(* LS Electric XG5000 project: AC1duobleanaloge *)
(* PLC NewPLC *)
(* module base 0 slot 0: Input/Output Module:XEC-DR60S (DC 24V INPUT 36points/RELAY OUTPUT 24points) *)
(* module base 0 slot 1: Input/Output Module:XBE-DR16A (DC 24V INPUT/RELAY OUTPUT, 16points) *)
(* module base 0 slot 2: Analog IO Module:XBF-AH04A (I/O, 2/2 CH) *)
(* module base 0 slot 9: Analog Output Module:XBO-DA02A (Volt/Current, 2-CH) *)
(* module base 0 slot 10: Analog Output Module:XBO-DA02A (Volt/Current, 2-CH) *)
VAR_GLOBAL
    _02_DA0_ACT AT %UX0.2.18 : BOOL; (* Analog IO Module: Output CH0 Active *)
    _02_DA0_DATA AT %UW0.2.7 : WORD; (* Analog IO Module: Output CH0 DATA *)
    _02_DA0_OUTEN AT %UX0.2.96 : BOOL; (* Analog IO Module: Output CH0 Status Setting *)
    _02_DA1_ACT AT %UX0.2.19 : BOOL; (* Analog IO Module: Output CH1 Active *)
    _02_DA1_DATA AT %UW0.2.8 : WORD; (* Analog IO Module: Output CH1 DATA *)
    _02_DA1_OUTEN AT %UX0.2.97 : BOOL; (* Analog IO Module: Output CH1 Status Setting *)
    _09_DA0_ACT AT %UX0.9.18 : BOOL; (* Analog Output Option Board: Output CH0 Active *)
    _09_DA0_OUTEN AT %UX0.9.96 : BOOL; (* Analog Output Option Board: Output CH0 Status Setting *)
    _09_DA1_ACT AT %UX0.9.19 : BOOL; (* Analog Output Option Board: Output CH1 Active *)
    _09_DA1_OUTEN AT %UX0.9.97 : BOOL; (* Analog Output Option Board: Output CH1 Status Setting *)
    _0A_DA0_ACT AT %UX0.10.18 : BOOL; (* Analog Output Option Board: Output CH0 Active *)
    _0A_DA0_OUTEN AT %UX0.10.96 : BOOL; (* Analog Output Option Board: Output CH0 Status Setting *)
    _0A_DA1_ACT AT %UX0.10.19 : BOOL; (* Analog Output Option Board: Output CH1 Active *)
    _0A_DA1_OUTEN AT %UX0.10.97 : BOOL; (* Analog Output Option Board: Output CH1 Status Setting *)
END_VAR

PROGRAM NewProgram_Copy (* task: Scan Program *)
VAR
    AAAA : WORD;
    aaaaaaaaaaaaaaa : REAL;
    acCONTROL AT %IX0.0.0 : BOOL;
    ACTRANS : BOOL;
    ADD1 : WORD;
    ADD2 : WORD;
    ANDOUT1 : WORD;
    AUTO AT %MX1 : BOOL;
    autoinhibit AT %MX222 : BOOL;
    BLOCK : UINT;
    chillerready : BOOL;
    COMPRESSOR : BOOL;
    CONTACTOR1 AT %QX0.0.0 : BOOL;
    CONTACTOR10 AT %QX0.0.9 : BOOL;
    CONTACTOR11 AT %QX0.0.20 : BOOL;
    CONTACTOR110 AT %IX0.0.29 : BOOL;
    CONTACTOR12 AT %QX0.0.21 : BOOL;
    CONTACTOR120 AT %IX0.0.30 : BOOL;
    CONTACTOR13 AT %QX0.0.22 : BOOL;
    CONTACTOR130 AT %IX0.0.31 : BOOL;
    CONTACTOR14 AT %QX0.0.23 : BOOL;
    CONTACTOR140 AT %IX0.0.32 : BOOL;
    CONTACTOR15 AT %QX0.1.0 : BOOL;
    CONTACTOR150 AT %IX0.0.33 : BOOL;
    CONTACTOR16 AT %QX0.1.1 : BOOL;
    CONTACTOR160 AT %IX0.0.34 : BOOL;
    CONTACTOR17 AT %QX0.1.2 : BOOL;
    CONTACTOR170 AT %IX0.1.1 : BOOL;
    CONTACTOR18 AT %QX0.1.3 : BOOL;
    CONTACTOR180 AT %IX0.1.0 : BOOL;
    CONTACTOR2 AT %QX0.0.1 : BOOL;
    CONTACTOR3 AT %QX0.0.2 : BOOL;
    CONTACTOR4 AT %QX0.0.3 : BOOL;
    CONTACTOR5 AT %QX0.0.4 : BOOL;
    CONTACTOR6 AT %QX0.0.5 : BOOL;
    CONTACTOR7 AT %QX0.0.6 : BOOL;
    CONTACTOR8 AT %QX0.0.7 : BOOL;
    CONTACTOR9 AT %QX0.0.8 : BOOL;
    CV : INT;
    damperon : BOOL;
    dcpower AT %IX0.0.1 : BOOL;
    DCPOWERK AT %QX0.1.4 : BOOL;
    dcpowerman AT %MX18 : BOOL;
    ddddddd : BOOL;
    DIV11 : WORD;
    DIV12 : INT;
    DIV124 : INT;
    DIV2 : WORD;
    DIV21 : WORD;
    DIV22 : WORD;
    DIV23 : WORD;
    DIV32 : INT;
    DIV33 : INT;
    DOOR1 AT %IX0.1.6 : BOOL;
    DOOR2 AT %IX0.1.7 : BOOL;
    DRIVE1ALARM AT %MX420 : BOOL;
    DRIVE2ALARM AT %MX421 : BOOL;
    DRIVEK1 AT %MX90 : BOOL;
    DRIVEK2 AT %MX91 : BOOL;
    DRIVEK3 : BOOL;
    DRIVEK4 : BOOL;
    DRIVEK5 : BOOL;
    DRIVEK6 : BOOL;
    DRIVEPUMP AT %MX92 : BOOL;
    dvi2 : DWORD;
    E11 : WORD;
    E2 : WORD;
    EE : WORD;
    EE1 : WORD;
    EE2 : WORD;
    ERR : BOOL;
    ET : TIME;
    FANREFSCALE : WORD;
    FANRUN : BOOL;
    FILTERRUN AT %MX50 : BOOL;
    FR10 AT %IX0.0.23 : BOOL;
    FR11 AT %IX0.0.24 : BOOL;
    FR12 AT %IX0.0.25 : BOOL;
    FR13 AT %IX0.0.26 : BOOL;
    FR14 AT %IX0.0.27 : BOOL;
    FR15 AT %IX0.0.28 : BOOL;
    FR8 AT %IX0.0.21 : BOOL;
    FR9 AT %IX0.0.22 : BOOL;
    HIMIDITYSCAL2 : WORD;
    HUMID2 : WORD;
    HUMID3 : WORD;
    HUMID4 : BOOL;
    HUMID5 : BOOL;
    HUMIDHIVALUE1 : WORD;
    HUMIDITIERR1 : WORD;
    HUMIDITYOUTSCAL : WORD;
    HUMIDLOWLIM1 : WORD;
    HUMIDNO1 : BOOL;
    HUMIDON : BOOL;
    hummidd : WORD;
    IN1 : SINT;
    IN10 : WORD;
    incin : WORD;
    inhumreal : REAL;
    inhumreal1 : REAL;
    inrealhuscale : REAL;
    inrealhuscale1 : REAL;
    INST : TON;
    INST1 : TON;
    INST10 : PIDRUN;
    INST11 : PIDRUN;
    INST12 : TON_UINT;
    INST13 : TON_UINT;
    INST14 : TON;
    INST15 : TON;
    INST16 : TON;
    INST17 : TON;
    INST18 : TON;
    INST19 : TON;
    INST2 : TON;
    INST20 : TON;
    INST21 : TON;
    INST22 : TON;
    INST23 : TON;
    INST24 : TON;
    INST25 : TON;
    INST26 : CTU_INT;
    INST27 : TON;
    INST28 : TON;
    INST29 : CTU_INT;
    INST3 : TON;
    INST30 : TON;
    INST31 : TON;
    INST32 : TON;
    INST33 : TON;
    INST34 : TON;
    INST35 : TON;
    INST36 : TON;
    INST37 : CTU_INT;
    INST38 : CTU_INT;
    INST39 : TON;
    INST4 : TON;
    INST40 : TON_UINT;
    INST41 : TON_UINT;
    INST42 : TON_UINT;
    INST43 : TON_UINT;
    INST44 : TON_UINT;
    INST45 : TON_UINT;
    INST46 : TON_UINT;
    INST47 : TMR;
    INST48 : TON_UINT;
    INST49 : TON_UINT;
    INST5 : TON;
    INST50 : TON_UINT;
    INST51 : TON_UINT;
    INST52 : TON_UINT;
    INST53 : TON;
    INST54 : TON;
    INST55 : TON;
    INST56 : TON;
    INST57 : TON;
    INST58 : TON;
    INST59 : TON;
    INST6 : TON;
    INST60 : TON;
    INST61 : TON;
    INST62 : CTU_INT;
    INST63 : CTR;
    INST64 : TON;
    INST65 : TON;
    INST66 : TON;
    INST67 : TON;
    INST68 : TON;
    INST69 : TON;
    INST7 : TON;
    INST70 : TON;
    INST71 : TON;
    INST72 : TON;
    INST73 : TON;
    INST74 : TON;
    INST75 : TON;
    INST76 : TON;
    INST77 : TON;
    INST8 : TON;
    INST9 : TON;
    K10ENDIS AT %MX129 : BOOL;
    K1B AT %MX95 : BOOL;
    k1endis AT %MX120 : BOOL;
    K2B AT %MX97 : BOOL;
    k2ENDIS AT %MX121 : BOOL;
    K3B : BOOL;
    K3ENDIS AT %MX122 : BOOL;
    K4B : BOOL;
    K4ENDIS AT %MX123 : BOOL;
    K5B : BOOL;
    K5ENDIS AT %MX124 : BOOL;
    K6B : BOOL;
    K6ENDIS AT %MX125 : BOOL;
    K7ENDIS AT %MX126 : BOOL;
    K8ENDIS AT %MX127 : BOOL;
    K9ENDIS AT %MX128 : BOOL;
    KDISCH1 AT %MX96 : BOOL;
    KDISCH2 : BOOL;
    KDISCH3 : BOOL;
    KSUC AT %MX94 : BOOL;
    KSUC2 : BOOL;
    KSUC3 : BOOL;
    LOOP : UINT;
    man1 : BOOL;
    man10 : BOOL;
    man2 : BOOL;
    man3 : BOOL;
    man4 : BOOL;
    man5 : BOOL;
    man6 : BOOL;
    man7 : BOOL;
    man8 : BOOL;
    man9 : BOOL;
    mot1 : BOOL;
    mot10 : BOOL;
    mot11 : BOOL;
    mot12 : BOOL;
    mot2 : BOOL;
    mot3 : BOOL;
    mot4 : BOOL;
    mot5 : BOOL;
    mot6 : BOOL;
    mot7 : BOOL;
    mot8 : BOOL;
    mot9 : BOOL;
    motor10 : BOOL;
    motor11 : BOOL;
    motor12 : BOOL;
    motor13 : BOOL;
    motor9 : BOOL;
    ooot : INT;
    OUT : SINT;
    OUT10 : INT;
    OUT100 : INT;
    OUT101 : REAL;
    OUT102 : REAL;
    OUT103 : INT;
    OUT104 : WORD;
    OUT20 : INT;
    OUT200 : WORD;
    out201 : INT;
    OUT202 : WORD;
    OUT203 : INT;
    OUT21 : INT;
    OUT300 : REAL;
    OUT301 : REAL;
    out310 : REAL;
    OUT351 : REAL;
    OUT352 : REAL;
    OUT50 : WORD;
    OUT6 : WORD;
    OUT6bit : BOOL;
    outhumreal : REAL;
    OUTrealhuscale : REAL;
    OUTTMP : WORD;
    OUTTMPLOWLIM : WORD;
    ouuu : INT;
    ouuuuuuut : DWORD;
    PID_STAT : WORD;
    PUMPON : BOOL;
    Q : BOOL;
    rstauto AT %MX2 : BOOL;
    RUNOK AT %MX98 : BOOL;
    scal11 : REAL;
    scale22 : REAL;
    scale23 : REAL;
    setauto AT %MX0 : BOOL;
    STATE1 : BOOL;
    STATE2 : BOOL;
    STATE3 : BOOL;
    STATE4 : BOOL;
    STATE5 : BOOL;
    STATE6 : BOOL;
    STATE7 : BOOL;
    step1 : BOOL;
    step10 : BOOL;
    step2 : BOOL;
    step3 : BOOL;
    step4 : BOOL;
    step5 : BOOL;
    step6 : BOOL;
    step7 : BOOL;
    step8 : BOOL;
    step9 : BOOL;
    SUCTION1RUN : BOOL;
    SUMMER : BOOL;
    teee : INT;
    TEMPE11 : WORD;
    TEMPLOWLIM1 : WORD;
    TEMPLOWLIM2 : INT;
    TEMPMAX1 : WORD;
    TEMPMAX2 : INT;
    VALVEACPOWER AT %QX0.1.7 : BOOL;
    VFD1 AT %QX0.0.10 : BOOL;
    VFD10 AT %QX0.0.19 : BOOL;
    VFD2 AT %QX0.0.11 : BOOL;
    VFD3 AT %QX0.0.12 : BOOL;
    VFD4 AT %QX0.0.13 : BOOL;
    VFD5 AT %QX0.0.14 : BOOL;
    VFD6 AT %QX0.0.15 : BOOL;
    VFD7 AT %QX0.0.16 : BOOL;
    VFD8 AT %QX0.0.17 : BOOL;
    VFD9 AT %QX0.0.18 : BOOL;
    WINTER : BOOL;
END_VAR
VAR RETAIN
    coldtemp AT %WW400 : INT;
    COLDTMP AT %WW240 : WORD;
    DIFFMAX AT %WW144 : WORD;
    DIFFMIN AT %WW142 : WORD;
    DIV1 : WORD;
    E1 AT %WW2004 : WORD;
    fanspeedhilim AT %WW156 : WORD;
    fanspeedlowlim AT %WW158 : WORD;
    FRESHDAMPER AT %WW310 : WORD;
    HIMIDITYSCALOUT AT %WW2016 : WORD;
    HOTTEMP AT %WW402 : INT;
    HOTTMP AT %WW230 : WORD;
    HUMIDHIVALUE AT %WW2012 : WORD;
    HUMIDINLEFTSENSOR AT %WW190 : WORD;
    HUMIDINRIGHTSENSOR AT %WW186 : WORD;
    HUMIDITIERR AT %WW2010 : WORD;
    HUMIDLOWLIM AT %WW2014 : WORD;
    HUMOUTSENSOR AT %WW184 : WORD;
    HUMSUM AT %WW178 : WORD;
    INHUMIDOFSET AT %WW177 : WORD;
    INHUMIDYSCALE AT %WW200 : WORD;
    INHUMIDYSCALE1 AT %WW204 : WORD;
    LEFTHUMIDSV AT %WW302 : WORD;
    MEANTEMP AT %WW520 : WORD;
    money AT %WW2800 : WORD;
    OUT5 AT %WW2008 : WORD;
    OUTHUMIDOFSET AT %WW179 : WORD;
    OUTHUMIDYSCALE AT %WW202 : WORD;
    OUTTEMP AT %WW210 : INT;
    pump1refrence AT %WW50 : WORD;
    pump2refrence AT %WW51 : WORD;
    rightHUMIDSV AT %WW300 : WORD;
    RIGHTZONFANREF AT %WW250 : WORD;
    scale1 AT %WD379 : REAL;
    scale2 AT %WD377 : REAL;
    SCALE21 AT %WD387 : REAL;
    temmmp AT %WW444 : WORD;
    TEMPE1 AT %WW2006 : WORD;
    TEMPINLEFTSENSOR AT %WW188 : WORD;
    TEMPINRIGHTSENSOR AT %WW185 : WORD;
    TEMPLOWLIM AT %WW2002 : INT;
    TEMPMAX AT %WW2000 : INT;
    TEMPOUTSESOR AT %WW183 : WORD;
    TEMPPV AT %WW220 : INT;
    TEMPPV1 AT %WW224 : INT;
    TEMPSV AT %WW10 : WORD;
    TEMPSV1 AT %WW12 : WORD;
    time1 AT %WW880 : WORD;
    timeout AT %WW890 : WORD;
END_VAR
VAR_EXTERNAL
    _02_DA0_ACT : BOOL; (* AT %UX0.2.18 *) (* Analog IO Module: Output CH0 Active *)
    _02_DA0_DATA : WORD; (* AT %UW0.2.7 *) (* Analog IO Module: Output CH0 DATA *)
    _02_DA0_OUTEN : BOOL; (* AT %UX0.2.96 *) (* Analog IO Module: Output CH0 Status Setting *)
    _02_DA1_ACT : BOOL; (* AT %UX0.2.19 *) (* Analog IO Module: Output CH1 Active *)
    _02_DA1_DATA : WORD; (* AT %UW0.2.8 *) (* Analog IO Module: Output CH1 DATA *)
    _02_DA1_OUTEN : BOOL; (* AT %UX0.2.97 *) (* Analog IO Module: Output CH1 Status Setting *)
    _09_DA0_ACT : BOOL; (* AT %UX0.9.18 *) (* Analog Output Option Board: Output CH0 Active *)
    _09_DA0_OUTEN : BOOL; (* AT %UX0.9.96 *) (* Analog Output Option Board: Output CH0 Status Setting *)
    _09_DA1_ACT : BOOL; (* AT %UX0.9.19 *) (* Analog Output Option Board: Output CH1 Active *)
    _09_DA1_OUTEN : BOOL; (* AT %UX0.9.97 *) (* Analog Output Option Board: Output CH1 Status Setting *)
    _0A_DA0_ACT : BOOL; (* AT %UX0.10.18 *) (* Analog Output Option Board: Output CH0 Active *)
    _0A_DA0_OUTEN : BOOL; (* AT %UX0.10.96 *) (* Analog Output Option Board: Output CH0 Status Setting *)
    _0A_DA1_ACT : BOOL; (* AT %UX0.10.19 *) (* Analog Output Option Board: Output CH1 Active *)
    _0A_DA1_OUTEN : BOOL; (* AT %UX0.10.97 *) (* Analog Output Option Board: Output CH1 Status Setting *)
END_VAR
VAR
    _e1 : R_TRIG;
    _e2 : R_TRIG;
    _e3 : R_TRIG;
    _e4 : F_TRIG;
    _e5 : R_TRIG;
    _e6 : R_TRIG;
    _e7 : R_TRIG;
    _p8 : BOOL;
    _e9 : R_TRIG;
    _t10 : BOOL;
    _e11 : R_TRIG;
    _e12 : F_TRIG;
    _t13 : BOOL;
    _t14 : BOOL;
    _t15 : BOOL;
    _t16 : BOOL;
    _t17 : BOOL;
    _t18 : BOOL;
    _t19 : BOOL;
    _t20 : BOOL;
    _t21 : BOOL;
    _t22 : BOOL;
    _t23 : BOOL;
    _t24 : BOOL;
    _t25 : BOOL;
    _t26 : BOOL;
    _t27 : BOOL;
    _t28 : BOOL;
    _t29 : BOOL;
    _t30 : BOOL;
    _t31 : BOOL;
    _t32 : BOOL;
    _t33 : BOOL;
    _t34 : BOOL;
    _t35 : BOOL;
    _t36 : BOOL;
    _t37 : BOOL;
END_VAR

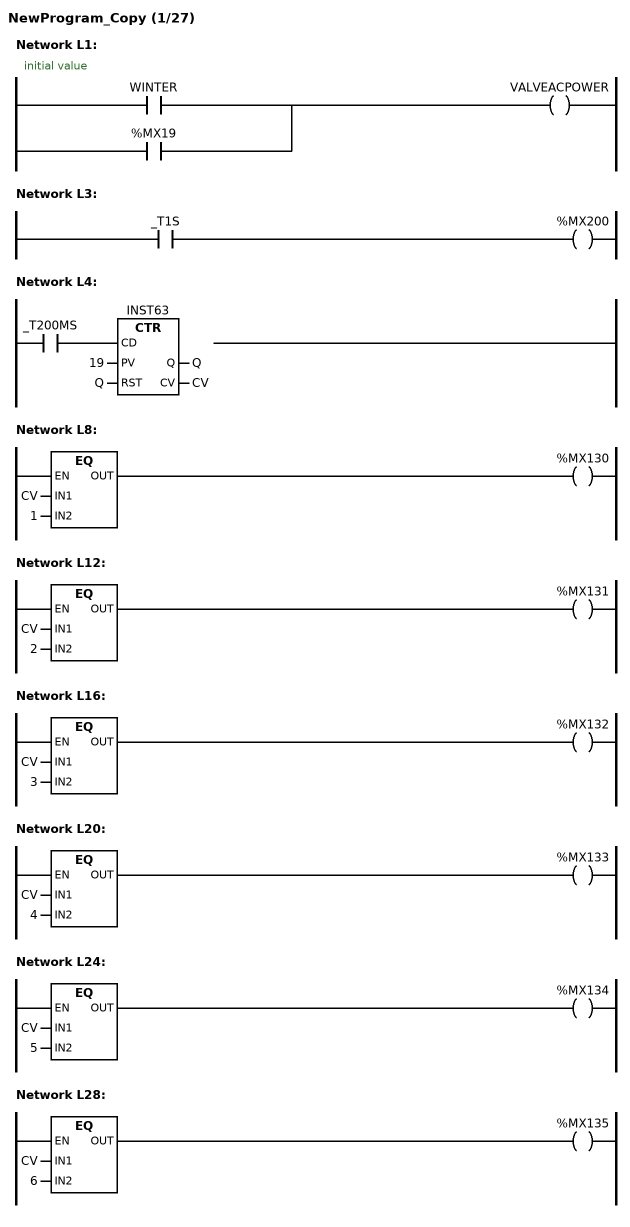
(* initial value *)
(* Rung L1 *)
VALVEACPOWER := WINTER OR %MX19;
(* Rung L3 *)
%MX200 := _T1S;
(* Rung L4 *)
INST63(CD := _T200MS, PV := 19, RST := Q, Q => Q, CV => CV);
(* Rung L8 *)
%MX130 := CV = 1;
(* Rung L12 *)
%MX131 := CV = 2;
(* Rung L16 *)
%MX132 := CV = 3;
(* Rung L20 *)
%MX133 := CV = 4;
(* Rung L24 *)
%MX134 := CV = 5;
(* Rung L28 *)
%MX135 := CV = 6;

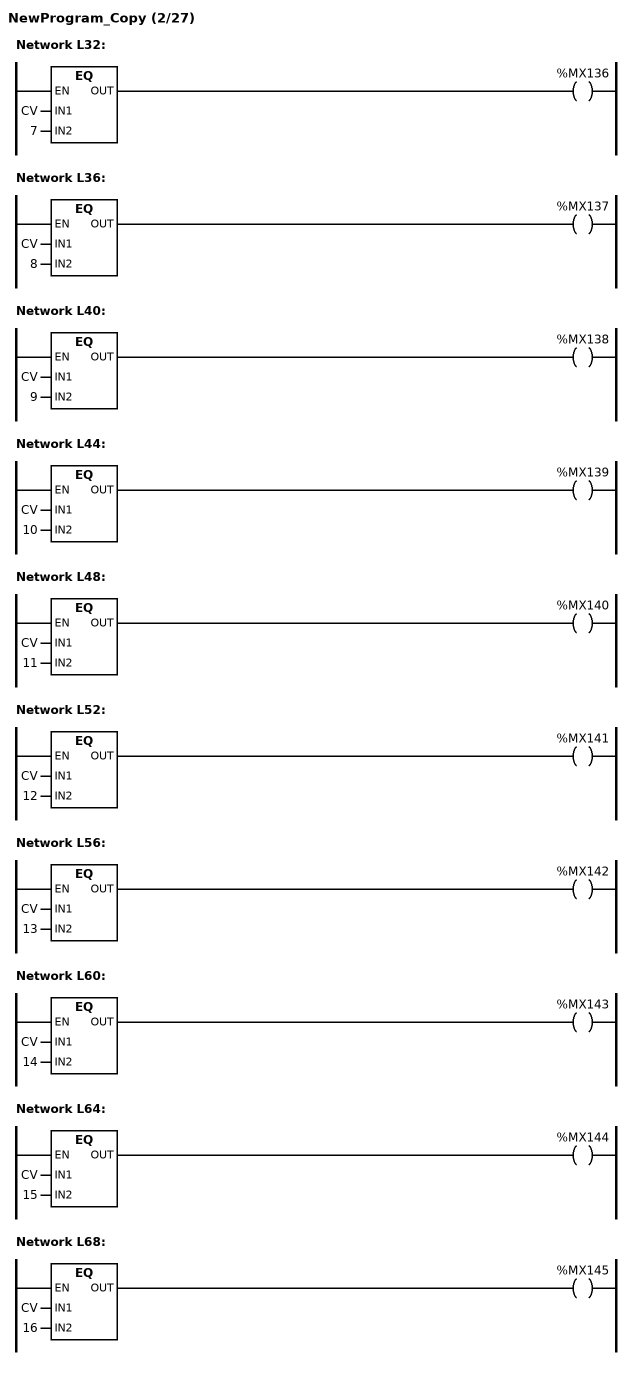
(* Rung L32 *)
%MX136 := CV = 7;
(* Rung L36 *)
%MX137 := CV = 8;
(* Rung L40 *)
%MX138 := CV = 9;
(* Rung L44 *)
%MX139 := CV = 10;
(* Rung L48 *)
%MX140 := CV = 11;
(* Rung L52 *)
%MX141 := CV = 12;
(* Rung L56 *)
%MX142 := CV = 13;
(* Rung L60 *)
%MX143 := CV = 14;
(* Rung L64 *)
%MX144 := CV = 15;
(* Rung L68 *)
%MX145 := CV = 16;

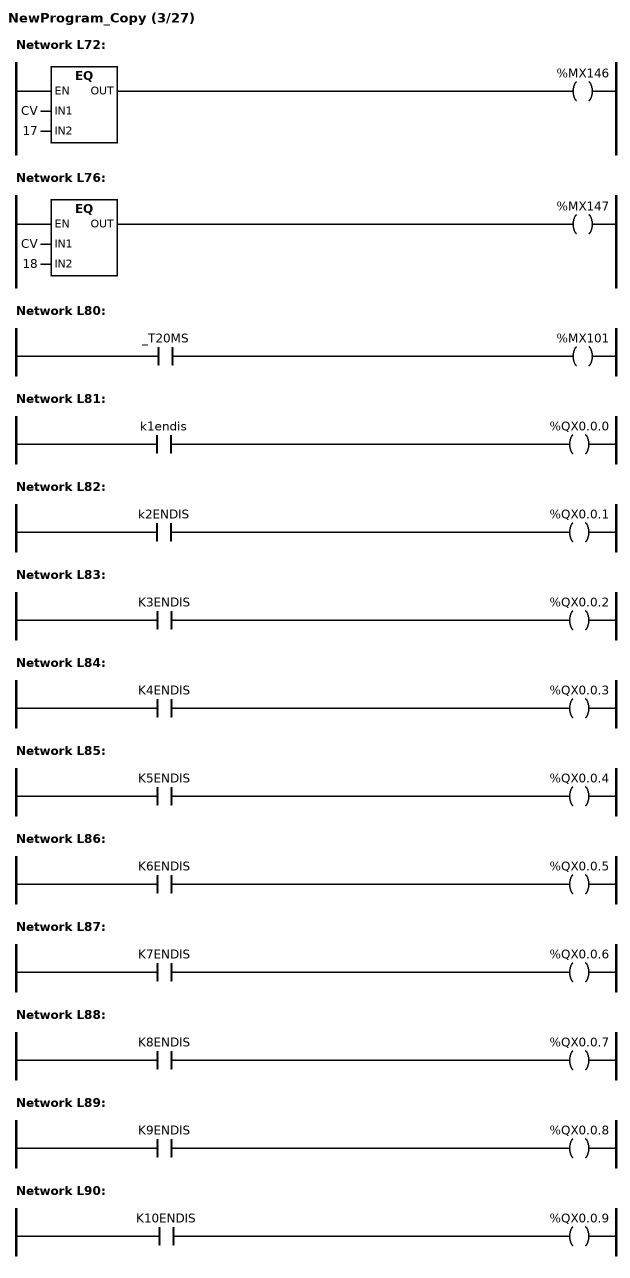
(* Rung L72 *)
%MX146 := CV = 17;
(* Rung L76 *)
%MX147 := CV = 18;
(* Rung L80 *)
%MX101 := _T20MS;
(* Rung L81 *)
%QX0.0.0 := k1endis;
(* Rung L82 *)
%QX0.0.1 := k2ENDIS;
(* Rung L83 *)
%QX0.0.2 := K3ENDIS;
(* Rung L84 *)
%QX0.0.3 := K4ENDIS;
(* Rung L85 *)
%QX0.0.4 := K5ENDIS;
(* Rung L86 *)
%QX0.0.5 := K6ENDIS;
(* Rung L87 *)
%QX0.0.6 := K7ENDIS;
(* Rung L88 *)
%QX0.0.7 := K8ENDIS;
(* Rung L89 *)
%QX0.0.8 := K9ENDIS;
(* Rung L90 *)
%QX0.0.9 := K10ENDIS;

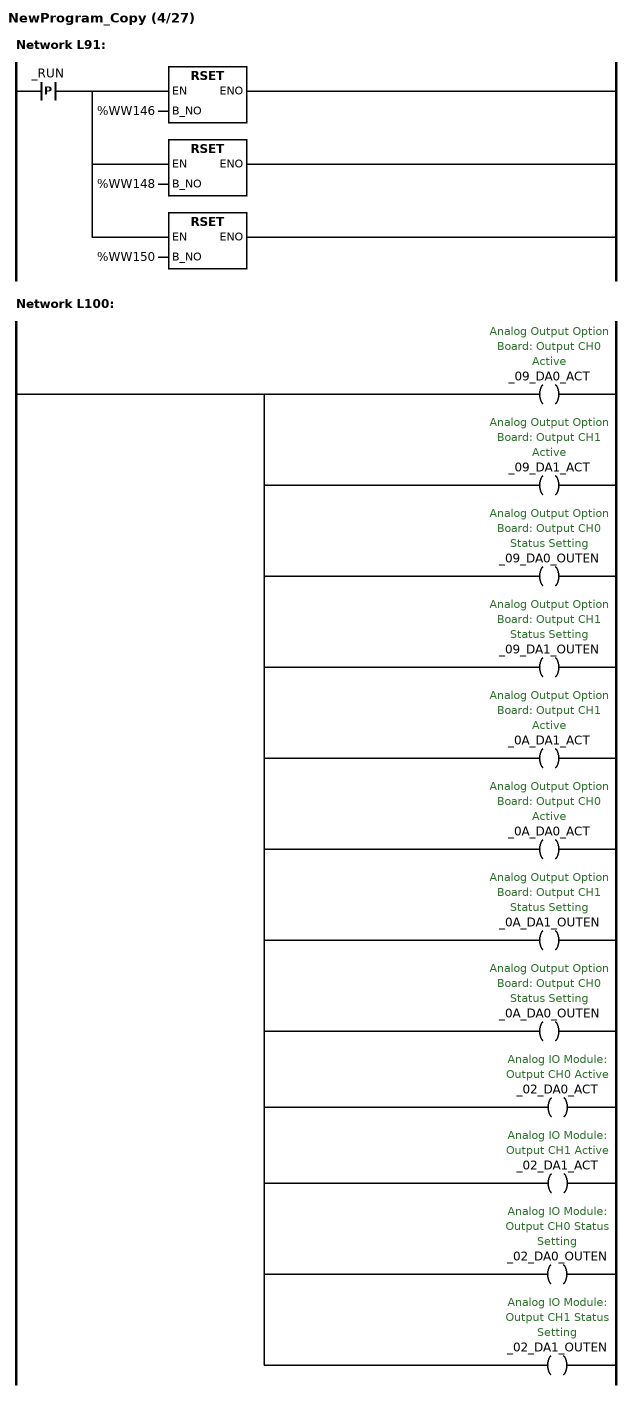
(* Rung L91 *)
_e1(CLK := _RUN);
IF _e1.Q THEN
    RSET(B_NO := %WW146);
    RSET(B_NO := %WW148);
    RSET(B_NO := %WW150);
END_IF;
(* Rung L100 *)
_09_DA0_ACT := TRUE;
_09_DA1_ACT := TRUE;
_09_DA0_OUTEN := TRUE;
_09_DA1_OUTEN := TRUE;
_0A_DA1_ACT := TRUE;
_0A_DA0_ACT := TRUE;
_0A_DA1_OUTEN := TRUE;
_0A_DA0_OUTEN := TRUE;
_02_DA0_ACT := TRUE;
_02_DA1_ACT := TRUE;
_02_DA0_OUTEN := TRUE;
_02_DA1_OUTEN := TRUE;

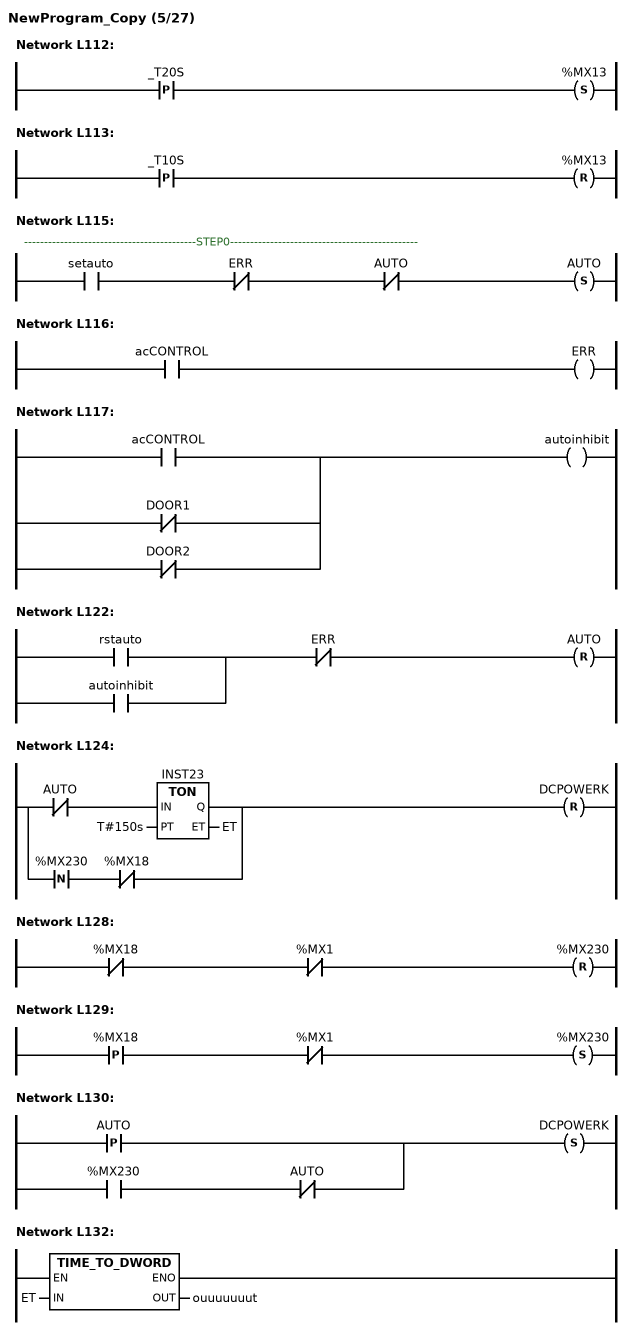
(* Rung L112 *)
_e2(CLK := _T20S);
IF _e2.Q THEN %MX13 := TRUE; END_IF;
(* Rung L113 *)
_e3(CLK := _T10S);
IF _e3.Q THEN %MX13 := FALSE; END_IF;
(* -------------------------------------------STEP0----------------------------------------------- *)
(* Rung L115 *)
IF setauto AND NOT ERR AND NOT AUTO THEN AUTO := TRUE; END_IF;
(* Rung L116 *)
ERR := acCONTROL;
(* Rung L117 *)
autoinhibit := acCONTROL OR NOT DOOR1 OR NOT DOOR2;
(* Rung L122 *)
IF (rstauto OR autoinhibit) AND NOT ERR THEN AUTO := FALSE; END_IF;
(* Rung L124 *)
INST23(IN := NOT AUTO, PT := T#150s, ET => ET);
_e4(CLK := %MX230);
IF INST23.Q OR (_e4.Q AND NOT %MX18) THEN DCPOWERK := FALSE; END_IF;
(* Rung L128 *)
IF NOT %MX18 AND NOT %MX1 THEN %MX230 := FALSE; END_IF;
(* Rung L129 *)
_e5(CLK := %MX18);
IF _e5.Q AND NOT %MX1 THEN %MX230 := TRUE; END_IF;
(* Rung L130 *)
_e6(CLK := AUTO);
IF _e6.Q OR (%MX230 AND NOT AUTO) THEN DCPOWERK := TRUE; END_IF;
(* Rung L132 *)
ouuuuuuut := TIME_TO_DWORD(ET);

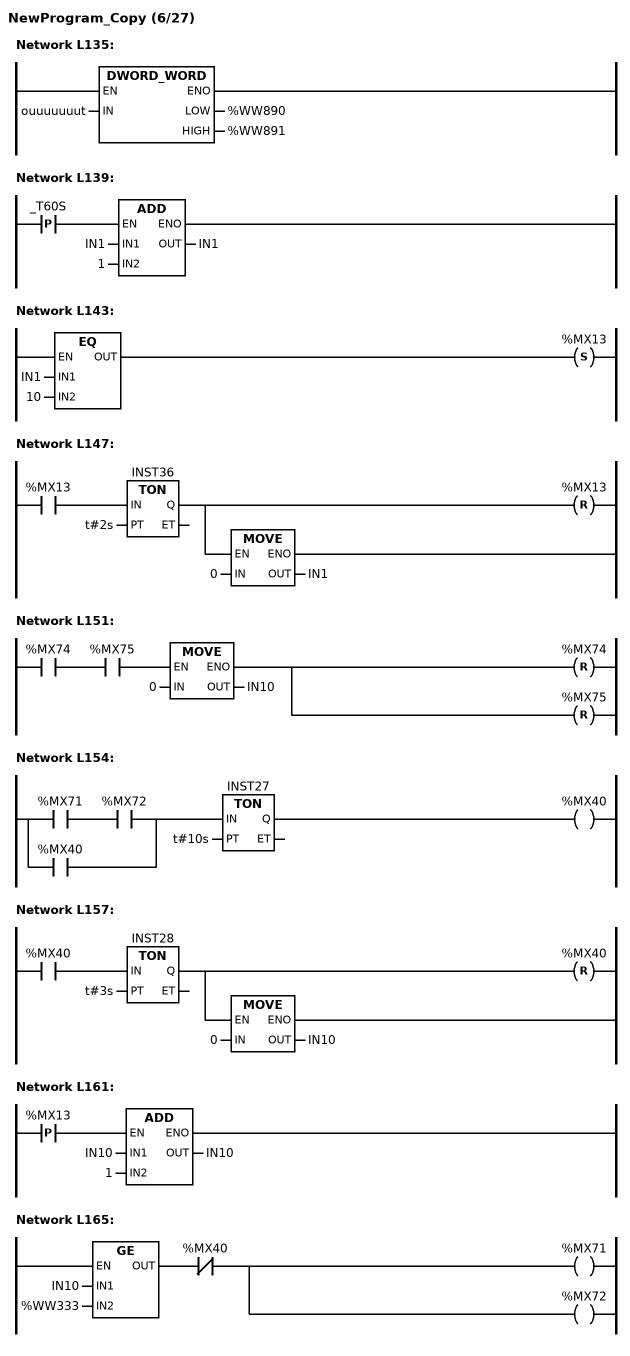
(* Rung L135 *)
%WW890 := DWORD_WORD(IN := ouuuuuuut, HIGH => %WW891);
(* Rung L139 *)
_e7(CLK := _T60S);
IF _e7.Q THEN IN1 := IN1 + 1; END_IF;
(* Rung L143 *)
IF IN1 = 10 THEN %MX13 := TRUE; END_IF;
(* Rung L147 *)
INST36(IN := %MX13, PT := t#2s);
IF INST36.Q THEN
    %MX13 := FALSE;
    IN1 := 0;
END_IF;
(* Rung L151 *)
IF %MX74 AND %MX75 THEN IN10 := 0; END_IF;
_p8 := %MX74 AND %MX75;
IF _p8 THEN
    %MX74 := FALSE;
    %MX75 := FALSE;
END_IF;
(* Rung L154 *)
INST27(IN := (%MX71 AND %MX72) OR %MX40, PT := t#10s);
%MX40 := INST27.Q;
(* Rung L157 *)
INST28(IN := %MX40, PT := t#3s);
IF INST28.Q THEN
    %MX40 := FALSE;
    IN10 := 0;
END_IF;
(* Rung L161 *)
_e9(CLK := %MX13);
IF _e9.Q THEN IN10 := IN10 + 1; END_IF;
(* Rung L165 *)
%MX71 := (IN10 >= %WW333) AND NOT %MX40;
%MX72 := (IN10 >= %WW333) AND NOT %MX40;

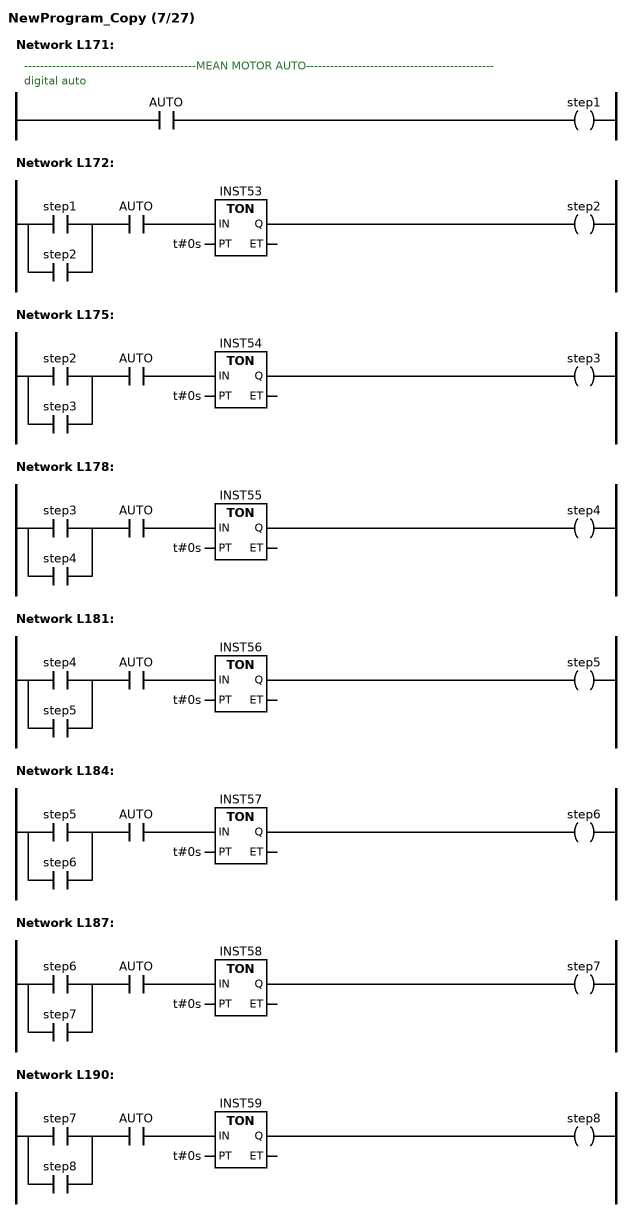
(* -------------------------------------------MEAN MOTOR AUTO----------------------------------------------- *)
(* digital auto *)
(* Rung L171 *)
step1 := AUTO;
(* Rung L172 *)
INST53(IN := (step1 OR step2) AND AUTO, PT := t#0s);
step2 := INST53.Q;
(* Rung L175 *)
INST54(IN := (step2 OR step3) AND AUTO, PT := t#0s);
step3 := INST54.Q;
(* Rung L178 *)
INST55(IN := (step3 OR step4) AND AUTO, PT := t#0s);
step4 := INST55.Q;
(* Rung L181 *)
INST56(IN := (step4 OR step5) AND AUTO, PT := t#0s);
step5 := INST56.Q;
(* Rung L184 *)
INST57(IN := (step5 OR step6) AND AUTO, PT := t#0s);
step6 := INST57.Q;
(* Rung L187 *)
INST58(IN := (step6 OR step7) AND AUTO, PT := t#0s);
step7 := INST58.Q;
(* Rung L190 *)
INST59(IN := (step7 OR step8) AND AUTO, PT := t#0s);
step8 := INST59.Q;

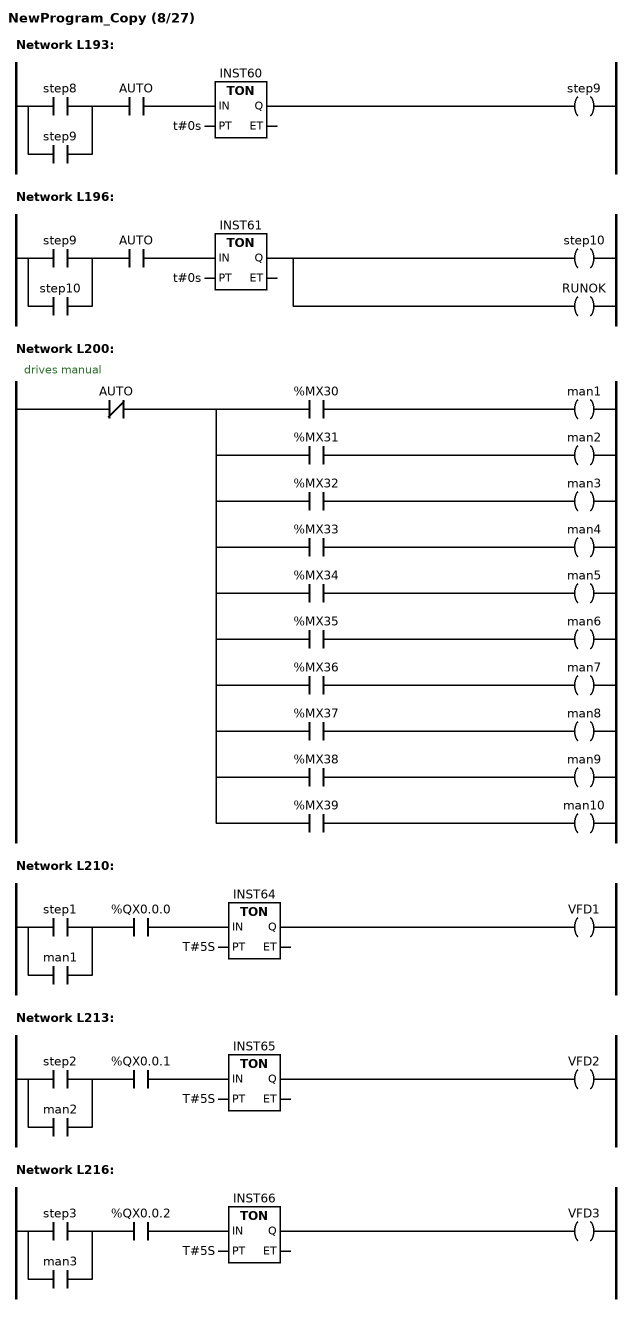
(* Rung L193 *)
INST60(IN := (step8 OR step9) AND AUTO, PT := t#0s);
step9 := INST60.Q;
(* Rung L196 *)
INST61(IN := (step9 OR step10) AND AUTO, PT := t#0s);
step10 := INST61.Q;
RUNOK := INST61.Q;
(* drives manual *)
(* Rung L200 *)
man1 := NOT AUTO AND %MX30;
man2 := NOT AUTO AND %MX31;
man3 := NOT AUTO AND %MX32;
man4 := NOT AUTO AND %MX33;
man5 := NOT AUTO AND %MX34;
man6 := NOT AUTO AND %MX35;
man7 := NOT AUTO AND %MX36;
man8 := NOT AUTO AND %MX37;
man9 := NOT AUTO AND %MX38;
man10 := NOT AUTO AND %MX39;
(* Rung L210 *)
INST64(IN := (step1 OR man1) AND %QX0.0.0, PT := T#5S);
VFD1 := INST64.Q;
(* Rung L213 *)
INST65(IN := (step2 OR man2) AND %QX0.0.1, PT := T#5S);
VFD2 := INST65.Q;
(* Rung L216 *)
INST66(IN := (step3 OR man3) AND %QX0.0.2, PT := T#5S);
VFD3 := INST66.Q;

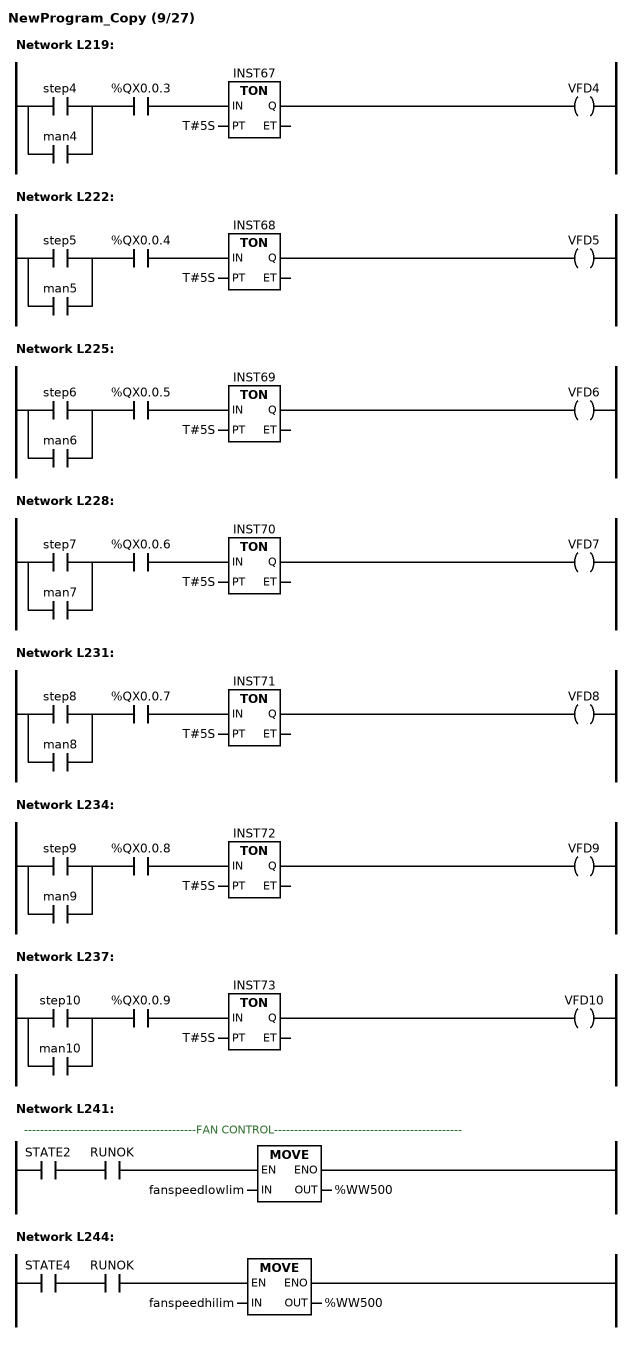
(* Rung L219 *)
INST67(IN := (step4 OR man4) AND %QX0.0.3, PT := T#5S);
VFD4 := INST67.Q;
(* Rung L222 *)
INST68(IN := (step5 OR man5) AND %QX0.0.4, PT := T#5S);
VFD5 := INST68.Q;
(* Rung L225 *)
INST69(IN := (step6 OR man6) AND %QX0.0.5, PT := T#5S);
VFD6 := INST69.Q;
(* Rung L228 *)
INST70(IN := (step7 OR man7) AND %QX0.0.6, PT := T#5S);
VFD7 := INST70.Q;
(* Rung L231 *)
INST71(IN := (step8 OR man8) AND %QX0.0.7, PT := T#5S);
VFD8 := INST71.Q;
(* Rung L234 *)
INST72(IN := (step9 OR man9) AND %QX0.0.8, PT := T#5S);
VFD9 := INST72.Q;
(* Rung L237 *)
INST73(IN := (step10 OR man10) AND %QX0.0.9, PT := T#5S);
VFD10 := INST73.Q;
(* -------------------------------------------FAN CONTROL----------------------------------------------- *)
(* Rung L241 *)
IF STATE2 AND RUNOK THEN %WW500 := fanspeedlowlim; END_IF;
(* Rung L244 *)
IF STATE4 AND RUNOK THEN %WW500 := fanspeedhilim; END_IF;

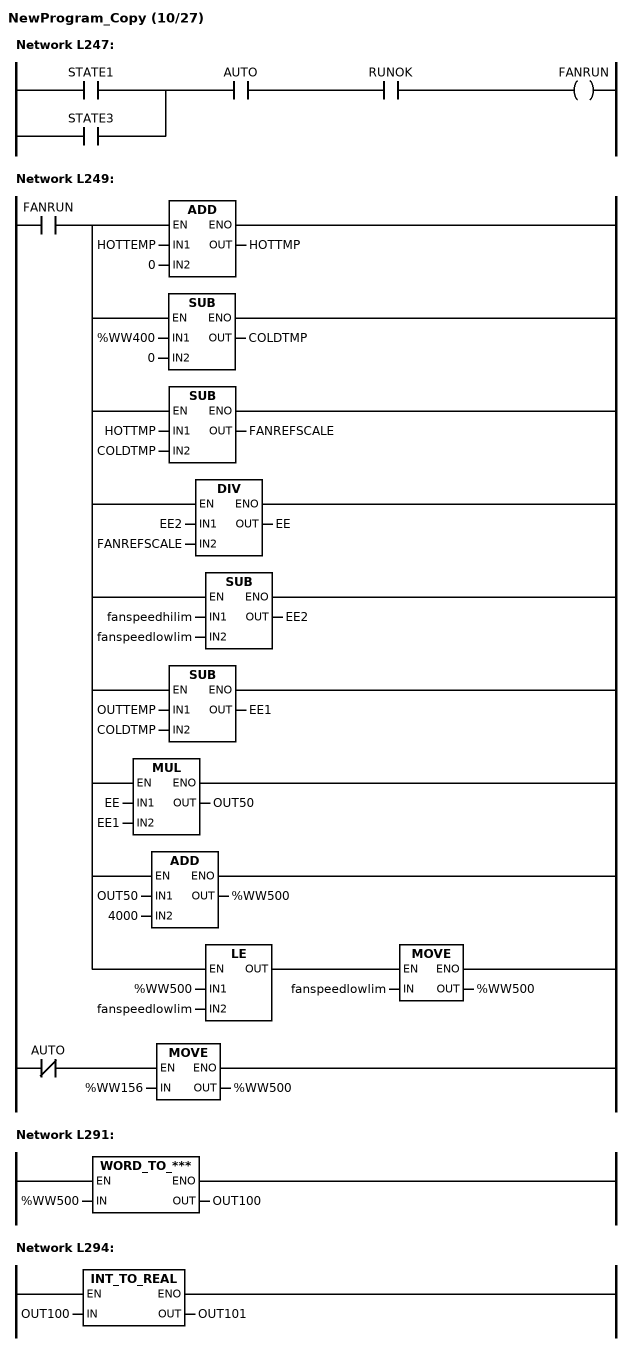
(* Rung L247 *)
FANRUN := (STATE1 OR STATE3) AND AUTO AND RUNOK;
(* Rung L249 *)
IF FANRUN THEN
    HOTTMP := HOTTEMP + 0;
    COLDTMP := %WW400 - 0;
    FANREFSCALE := HOTTMP - COLDTMP;
    EE := EE2 / FANREFSCALE;
    EE2 := fanspeedhilim - fanspeedlowlim;
    EE1 := OUTTEMP - COLDTMP;
    OUT50 := EE * EE1;
    %WW500 := OUT50 + 4000;
    _t10 := %WW500 <= fanspeedlowlim;
END_IF;
IF _t10 THEN %WW500 := fanspeedlowlim; END_IF;
IF NOT AUTO THEN %WW500 := %WW156; END_IF;
(* Rung L291 *)
OUT100 := WORD_TO_***(%WW500);
(* Rung L294 *)
OUT101 := INT_TO_REAL(OUT100);

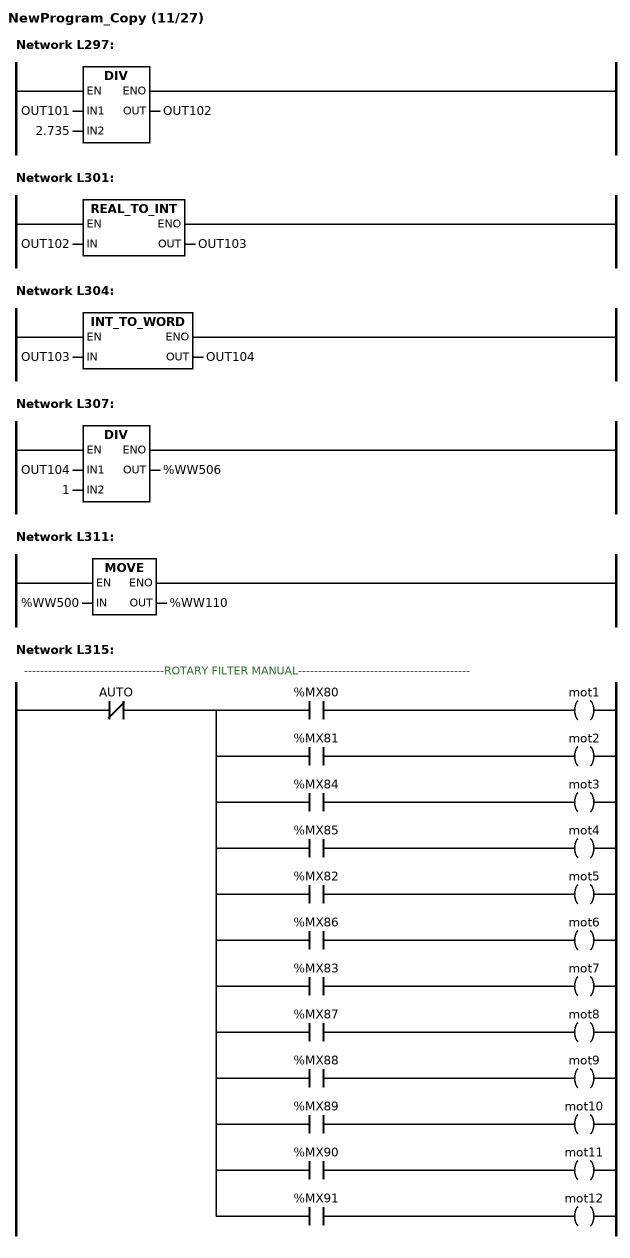
(* Rung L297 *)
OUT102 := OUT101 / 2.735;
(* Rung L301 *)
OUT103 := REAL_TO_INT(OUT102);
(* Rung L304 *)
OUT104 := INT_TO_WORD(OUT103);
(* Rung L307 *)
%WW506 := OUT104 / 1;
(* Rung L311 *)
%WW110 := %WW500;
(* -----------------------------------ROTARY FILTER MANUAL------------------------------------------- *)
(* Rung L315 *)
mot1 := NOT AUTO AND %MX80;
mot2 := NOT AUTO AND %MX81;
mot3 := NOT AUTO AND %MX84;
mot4 := NOT AUTO AND %MX85;
mot5 := NOT AUTO AND %MX82;
mot6 := NOT AUTO AND %MX86;
mot7 := NOT AUTO AND %MX83;
mot8 := NOT AUTO AND %MX87;
mot9 := NOT AUTO AND %MX88;
mot10 := NOT AUTO AND %MX89;
mot11 := NOT AUTO AND %MX90;
mot12 := NOT AUTO AND %MX91;

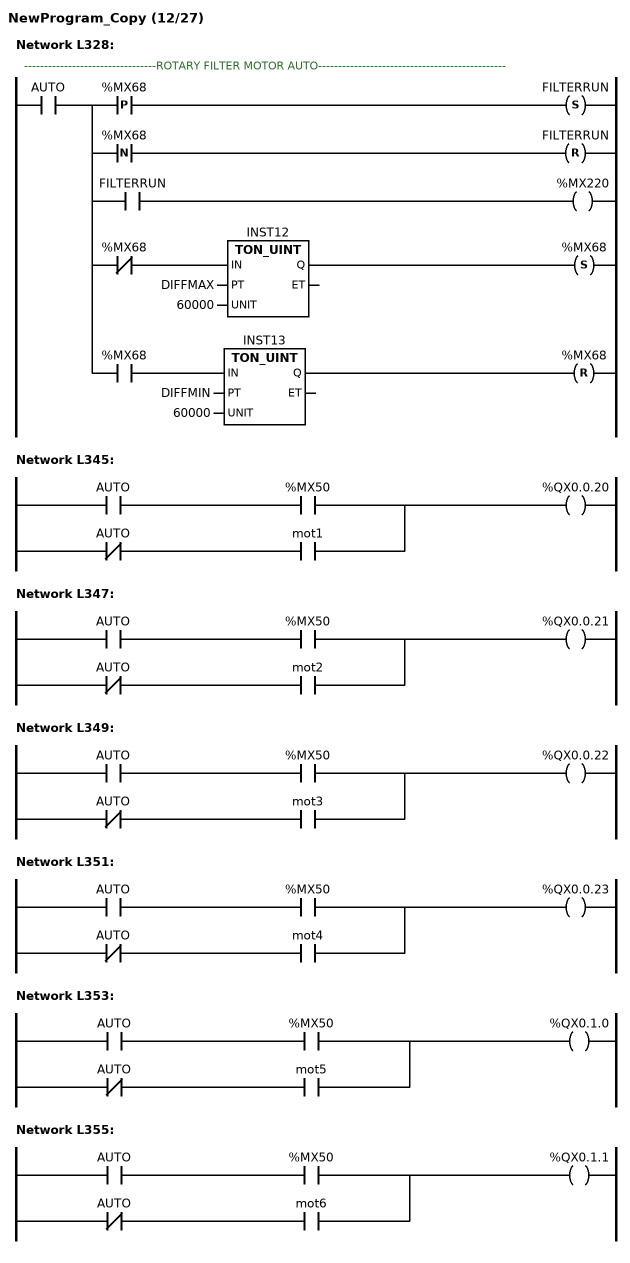
(* ---------------------------------ROTARY FILTER MOTOR AUTO----------------------------------------------- *)
(* Rung L328 *)
_e11(CLK := %MX68);
IF AUTO AND _e11.Q THEN FILTERRUN := TRUE; END_IF;
_e12(CLK := %MX68);
IF AUTO AND _e12.Q THEN FILTERRUN := FALSE; END_IF;
%MX220 := AUTO AND FILTERRUN;
INST12(IN := AUTO AND NOT %MX68, PT := DIFFMAX, UNIT := 60000);
IF INST12.Q THEN %MX68 := TRUE; END_IF;
INST13(IN := AUTO AND %MX68, PT := DIFFMIN, UNIT := 60000);
IF INST13.Q THEN %MX68 := FALSE; END_IF;
(* Rung L345 *)
%QX0.0.20 := (AUTO AND %MX50) OR (NOT AUTO AND mot1);
(* Rung L347 *)
%QX0.0.21 := (AUTO AND %MX50) OR (NOT AUTO AND mot2);
(* Rung L349 *)
%QX0.0.22 := (AUTO AND %MX50) OR (NOT AUTO AND mot3);
(* Rung L351 *)
%QX0.0.23 := (AUTO AND %MX50) OR (NOT AUTO AND mot4);
(* Rung L353 *)
%QX0.1.0 := (AUTO AND %MX50) OR (NOT AUTO AND mot5);
(* Rung L355 *)
%QX0.1.1 := (AUTO AND %MX50) OR (NOT AUTO AND mot6);

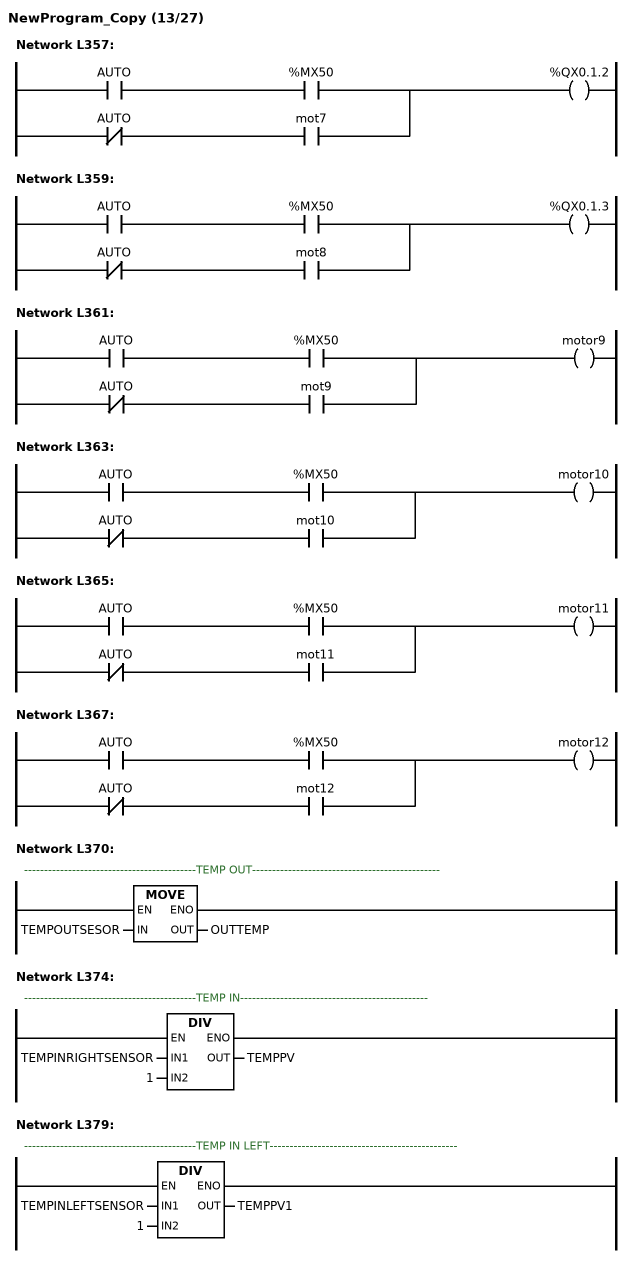
(* Rung L357 *)
%QX0.1.2 := (AUTO AND %MX50) OR (NOT AUTO AND mot7);
(* Rung L359 *)
%QX0.1.3 := (AUTO AND %MX50) OR (NOT AUTO AND mot8);
(* Rung L361 *)
motor9 := (AUTO AND %MX50) OR (NOT AUTO AND mot9);
(* Rung L363 *)
motor10 := (AUTO AND %MX50) OR (NOT AUTO AND mot10);
(* Rung L365 *)
motor11 := (AUTO AND %MX50) OR (NOT AUTO AND mot11);
(* Rung L367 *)
motor12 := (AUTO AND %MX50) OR (NOT AUTO AND mot12);
(* -------------------------------------------TEMP OUT----------------------------------------------- *)
(* Rung L370 *)
OUTTEMP := TEMPOUTSESOR;
(* -------------------------------------------TEMP IN----------------------------------------------- *)
(* Rung L374 *)
TEMPPV := TEMPINRIGHTSENSOR / 1;
(* -------------------------------------------TEMP IN LEFT----------------------------------------------- *)
(* Rung L379 *)
TEMPPV1 := TEMPINLEFTSENSOR / 1;

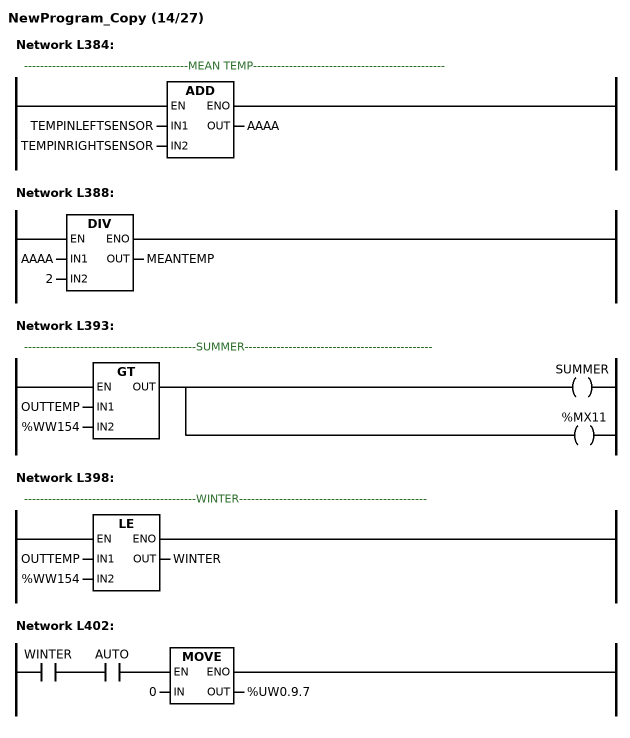
(* -----------------------------------------MEAN TEMP------------------------------------------------ *)
(* Rung L384 *)
AAAA := TEMPINLEFTSENSOR + TEMPINRIGHTSENSOR;
(* Rung L388 *)
MEANTEMP := AAAA / 2;
(* -------------------------------------------SUMMER----------------------------------------------- *)
(* Rung L393 *)
SUMMER := OUTTEMP > %WW154;
%MX11 := OUTTEMP > %WW154;
(* -------------------------------------------WINTER----------------------------------------------- *)
(* Rung L398 *)
WINTER := OUTTEMP <= %WW154;
(* Rung L402 *)
IF WINTER AND AUTO THEN %UW0.9.7 := 0; END_IF;

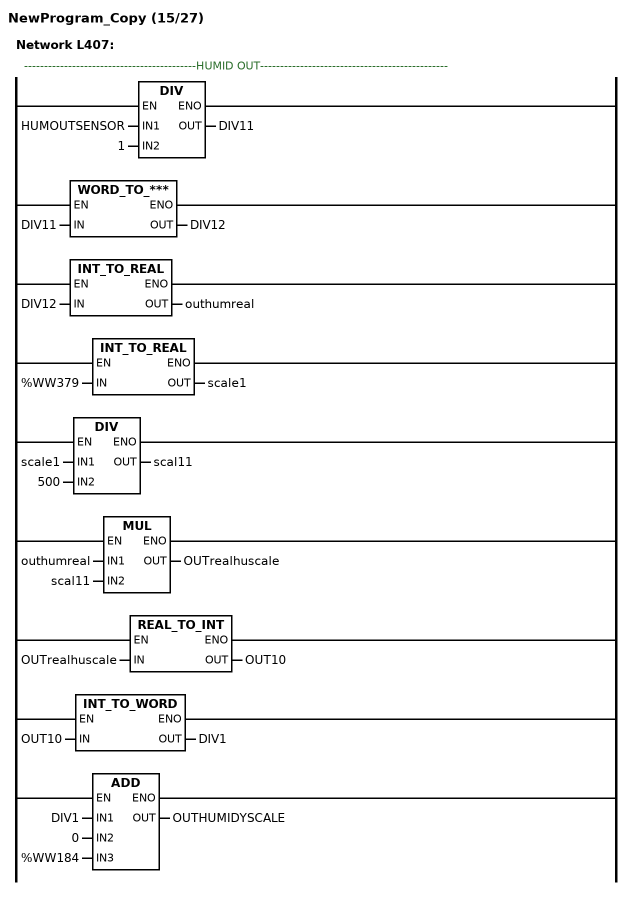
(* -------------------------------------------HUMID OUT----------------------------------------------- *)
(* Rung L407 *)
DIV11 := HUMOUTSENSOR / 1;
DIV12 := WORD_TO_***(DIV11);
outhumreal := INT_TO_REAL(DIV12);
scale1 := INT_TO_REAL(%WW379);
scal11 := scale1 / 500;
OUTrealhuscale := outhumreal * scal11;
OUT10 := REAL_TO_INT(OUTrealhuscale);
DIV1 := INT_TO_WORD(OUT10);
OUTHUMIDYSCALE := DIV1 + 0 + %WW184;

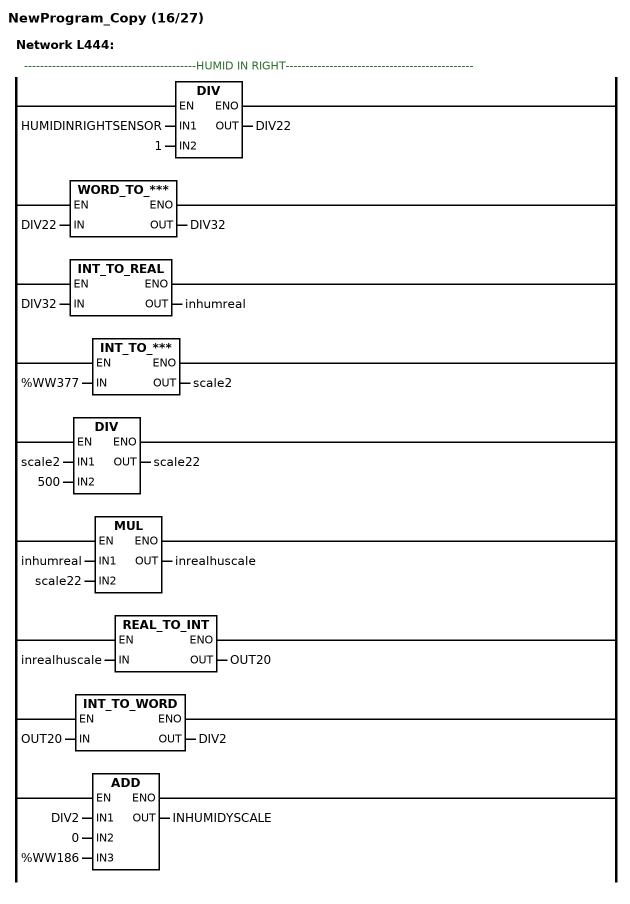
(* -------------------------------------------HUMID IN RIGHT----------------------------------------------- *)
(* Rung L444 *)
DIV22 := HUMIDINRIGHTSENSOR / 1;
DIV32 := WORD_TO_***(DIV22);
inhumreal := INT_TO_REAL(DIV32);
scale2 := INT_TO_***(%WW377);
scale22 := scale2 / 500;
inrealhuscale := inhumreal * scale22;
OUT20 := REAL_TO_INT(inrealhuscale);
DIV2 := INT_TO_WORD(OUT20);
INHUMIDYSCALE := DIV2 + 0 + %WW186;

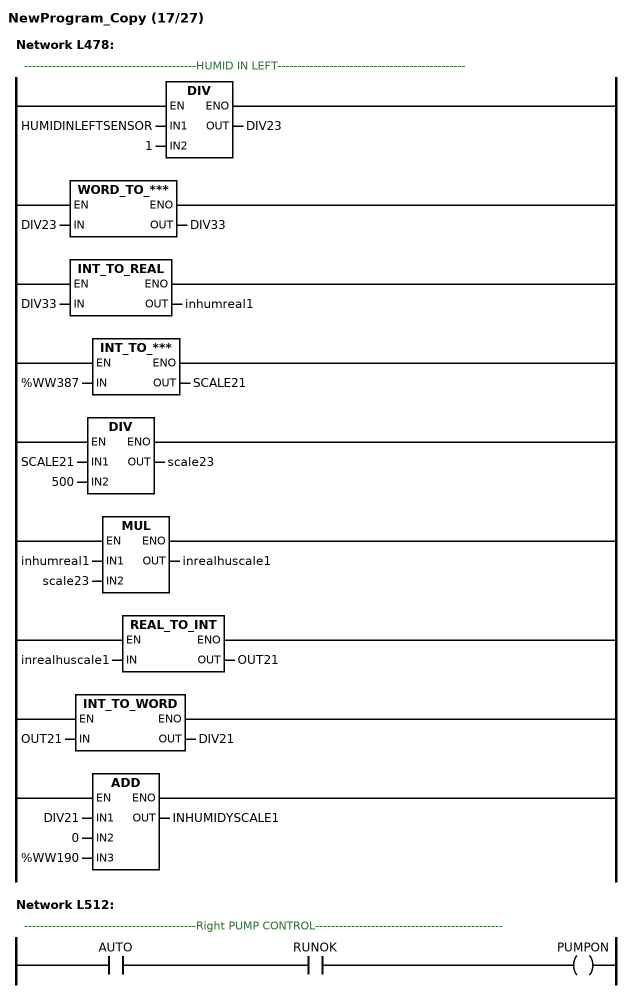
(* -------------------------------------------HUMID IN LEFT----------------------------------------------- *)
(* Rung L478 *)
DIV23 := HUMIDINLEFTSENSOR / 1;
DIV33 := WORD_TO_***(DIV23);
inhumreal1 := INT_TO_REAL(DIV33);
SCALE21 := INT_TO_***(%WW387);
scale23 := SCALE21 / 500;
inrealhuscale1 := inhumreal1 * scale23;
OUT21 := REAL_TO_INT(inrealhuscale1);
DIV21 := INT_TO_WORD(OUT21);
INHUMIDYSCALE1 := DIV21 + 0 + %WW190;
(* -------------------------------------------Right PUMP CONTROL----------------------------------------------- *)
(* Rung L512 *)
PUMPON := AUTO AND RUNOK;

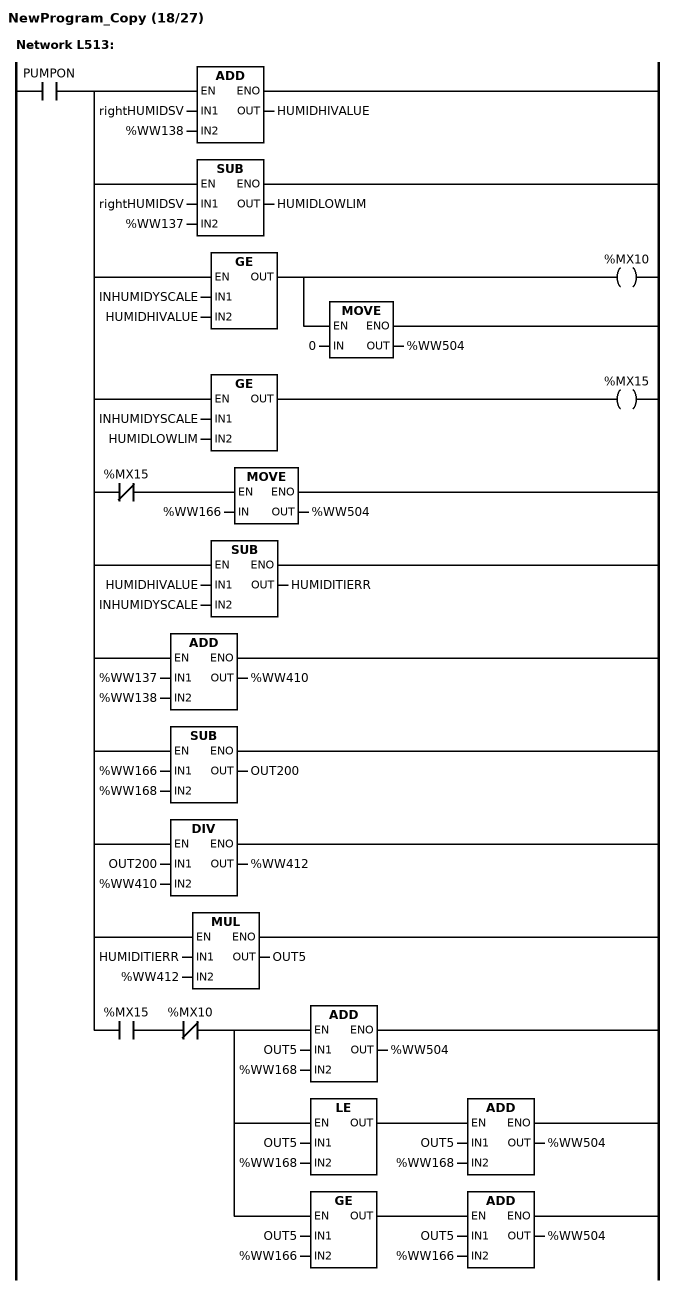
(* Rung L513 *)
IF PUMPON THEN
    HUMIDHIVALUE := rightHUMIDSV + %WW138;
    HUMIDLOWLIM := rightHUMIDSV - %WW137;
    _t13 := INHUMIDYSCALE >= HUMIDHIVALUE;
END_IF;
%MX10 := _t13;
IF _t13 THEN %WW504 := 0; END_IF;
IF PUMPON THEN _t14 := INHUMIDYSCALE >= HUMIDLOWLIM; END_IF;
%MX15 := _t14;
IF PUMPON AND NOT %MX15 THEN %WW504 := %WW166; END_IF;
IF PUMPON THEN
    HUMIDITIERR := HUMIDHIVALUE - INHUMIDYSCALE;
    %WW410 := %WW137 + %WW138;
    OUT200 := %WW166 - %WW168;
    %WW412 := OUT200 / %WW410;
    OUT5 := HUMIDITIERR * %WW412;
END_IF;
IF PUMPON AND %MX15 AND NOT %MX10 THEN
    %WW504 := OUT5 + %WW168;
    _t15 := OUT5 <= %WW168;
END_IF;
IF _t15 THEN %WW504 := OUT5 + %WW168; END_IF;
IF PUMPON AND %MX15 AND NOT %MX10 THEN _t16 := OUT5 >= %WW166; END_IF;
IF _t16 THEN %WW504 := OUT5 + %WW166; END_IF;

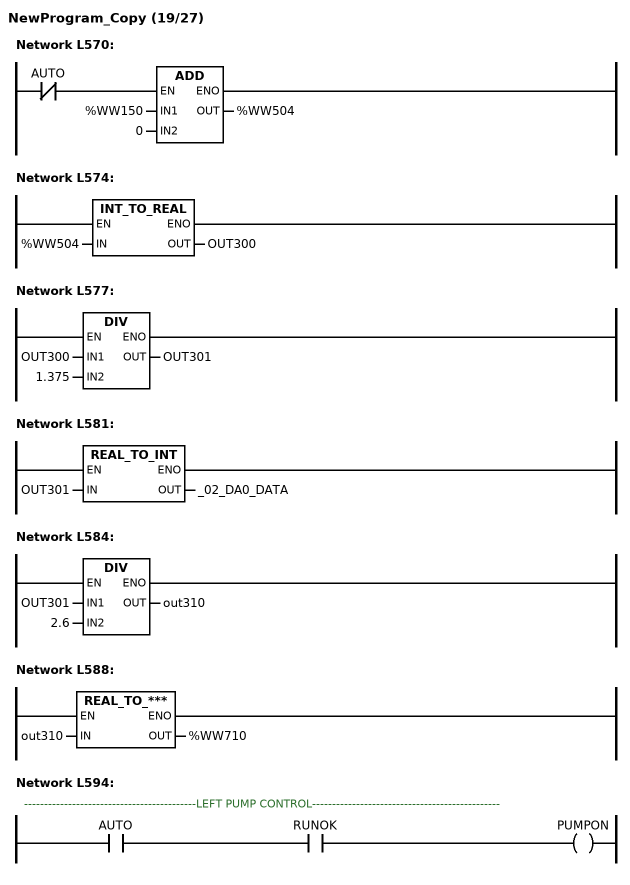
(* Rung L570 *)
IF NOT AUTO THEN %WW504 := %WW150 + 0; END_IF;
(* Rung L574 *)
OUT300 := INT_TO_REAL(%WW504);
(* Rung L577 *)
OUT301 := OUT300 / 1.375;
(* Rung L581 *)
_02_DA0_DATA := REAL_TO_INT(OUT301);
(* Rung L584 *)
out310 := OUT301 / 2.6;
(* Rung L588 *)
%WW710 := REAL_TO_***(out310);
(* -------------------------------------------LEFT PUMP CONTROL----------------------------------------------- *)
(* Rung L594 *)
PUMPON := AUTO AND RUNOK;

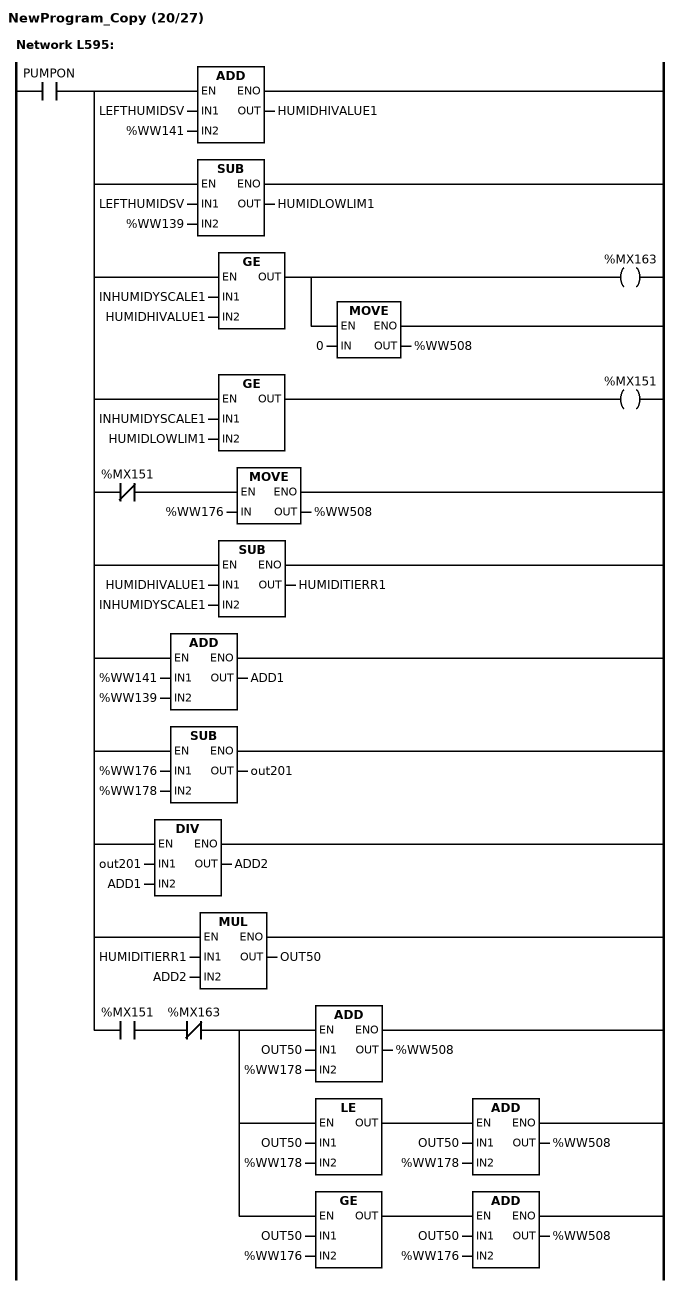
(* Rung L595 *)
IF PUMPON THEN
    HUMIDHIVALUE1 := LEFTHUMIDSV + %WW141;
    HUMIDLOWLIM1 := LEFTHUMIDSV - %WW139;
    _t17 := INHUMIDYSCALE1 >= HUMIDHIVALUE1;
END_IF;
%MX163 := _t17;
IF _t17 THEN %WW508 := 0; END_IF;
IF PUMPON THEN _t18 := INHUMIDYSCALE1 >= HUMIDLOWLIM1; END_IF;
%MX151 := _t18;
IF PUMPON AND NOT %MX151 THEN %WW508 := %WW176; END_IF;
IF PUMPON THEN
    HUMIDITIERR1 := HUMIDHIVALUE1 - INHUMIDYSCALE1;
    ADD1 := %WW141 + %WW139;
    out201 := %WW176 - %WW178;
    ADD2 := out201 / ADD1;
    OUT50 := HUMIDITIERR1 * ADD2;
END_IF;
IF PUMPON AND %MX151 AND NOT %MX163 THEN
    %WW508 := OUT50 + %WW178;
    _t19 := OUT50 <= %WW178;
END_IF;
IF _t19 THEN %WW508 := OUT50 + %WW178; END_IF;
IF PUMPON AND %MX151 AND NOT %MX163 THEN _t20 := OUT50 >= %WW176; END_IF;
IF _t20 THEN %WW508 := OUT50 + %WW176; END_IF;

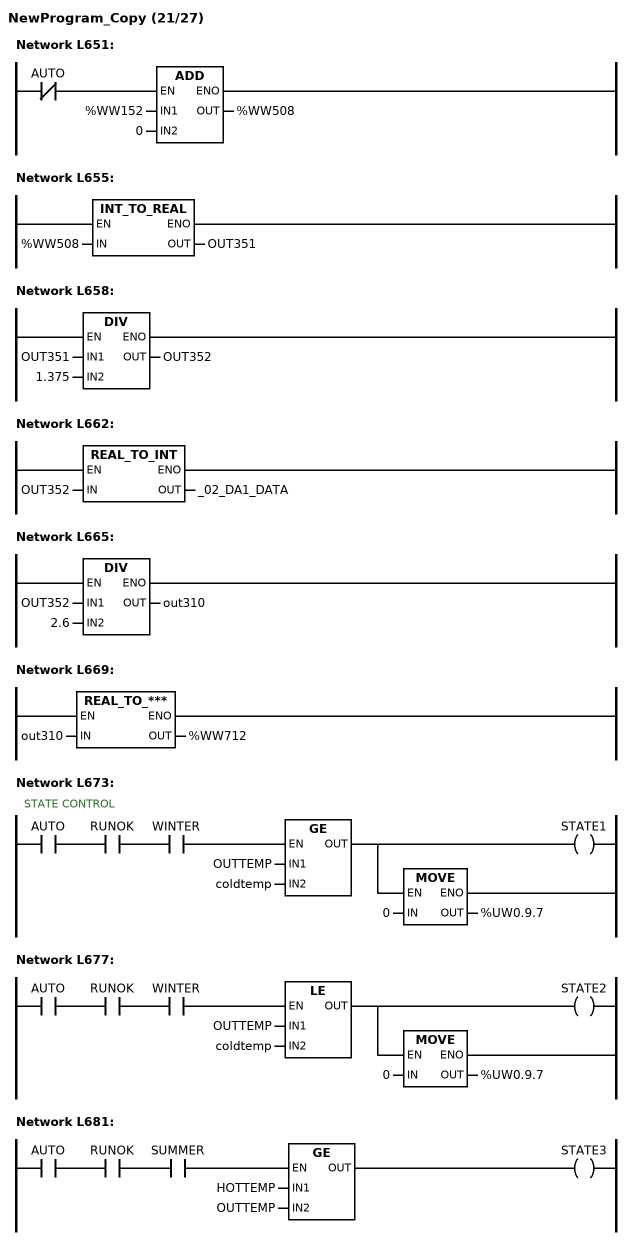
(* Rung L651 *)
IF NOT AUTO THEN %WW508 := %WW152 + 0; END_IF;
(* Rung L655 *)
OUT351 := INT_TO_REAL(%WW508);
(* Rung L658 *)
OUT352 := OUT351 / 1.375;
(* Rung L662 *)
_02_DA1_DATA := REAL_TO_INT(OUT352);
(* Rung L665 *)
out310 := OUT352 / 2.6;
(* Rung L669 *)
%WW712 := REAL_TO_***(out310);
(* STATE CONTROL *)
(* Rung L673 *)
IF AUTO AND RUNOK AND WINTER THEN _t21 := OUTTEMP >= coldtemp; END_IF;
STATE1 := _t21;
IF _t21 THEN %UW0.9.7 := 0; END_IF;
(* Rung L677 *)
IF AUTO AND RUNOK AND WINTER THEN _t22 := OUTTEMP <= coldtemp; END_IF;
STATE2 := _t22;
IF _t22 THEN %UW0.9.7 := 0; END_IF;
(* Rung L681 *)
IF AUTO AND RUNOK AND SUMMER THEN _t23 := HOTTEMP >= OUTTEMP; END_IF;
STATE3 := _t23;

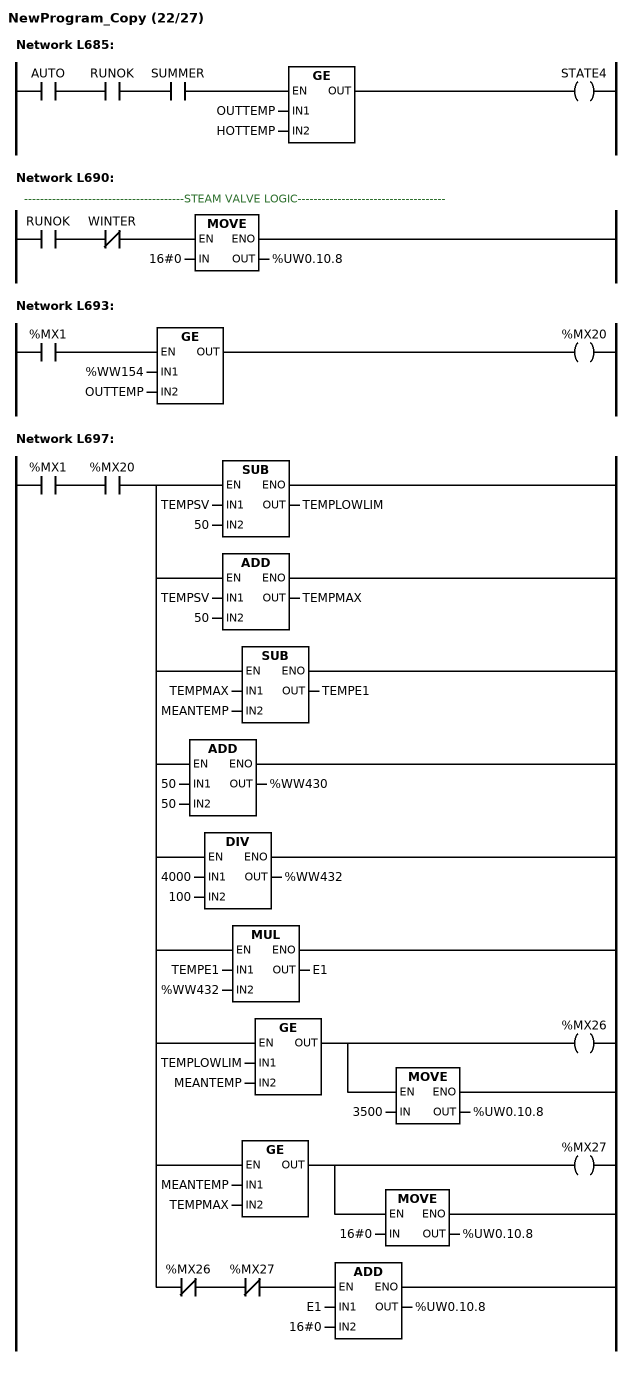
(* Rung L685 *)
IF AUTO AND RUNOK AND SUMMER THEN _t24 := OUTTEMP >= HOTTEMP; END_IF;
STATE4 := _t24;
(* ----------------------------------------STEAM VALVE LOGIC------------------------------------- *)
(* Rung L690 *)
IF RUNOK AND NOT WINTER THEN %UW0.10.8 := 16#0; END_IF;
(* Rung L693 *)
IF %MX1 THEN _t25 := %WW154 >= OUTTEMP; END_IF;
%MX20 := _t25;
(* Rung L697 *)
IF %MX1 AND %MX20 THEN
    TEMPLOWLIM := TEMPSV - 50;
    TEMPMAX := TEMPSV + 50;
    TEMPE1 := TEMPMAX - MEANTEMP;
    %WW430 := 50 + 50;
    %WW432 := 4000 / 100;
    E1 := TEMPE1 * %WW432;
    _t26 := TEMPLOWLIM >= MEANTEMP;
END_IF;
%MX26 := _t26;
IF _t26 THEN %UW0.10.8 := 3500; END_IF;
IF %MX1 AND %MX20 THEN _t27 := MEANTEMP >= TEMPMAX; END_IF;
%MX27 := _t27;
IF _t27 THEN %UW0.10.8 := 16#0; END_IF;
IF %MX1 AND %MX20 AND NOT %MX26 AND NOT %MX27 THEN %UW0.10.8 := E1 + 16#0; END_IF;

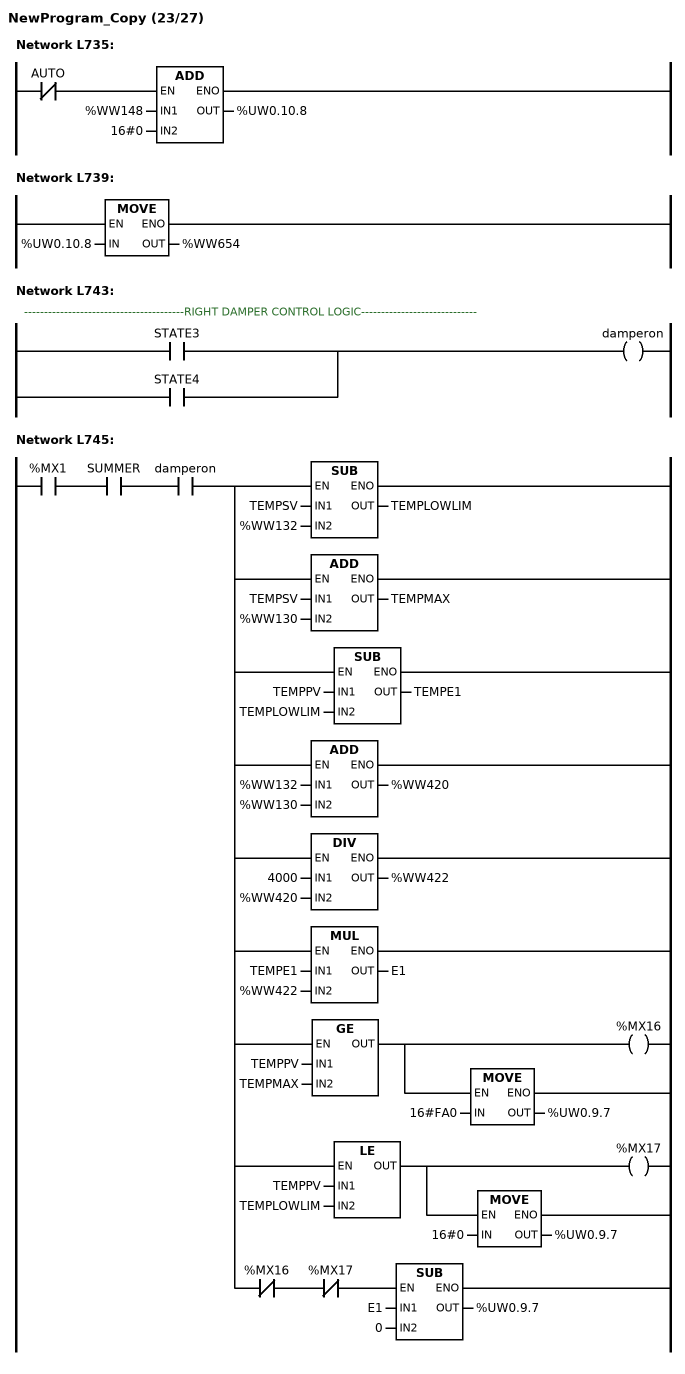
(* Rung L735 *)
IF NOT AUTO THEN %UW0.10.8 := %WW148 + 16#0; END_IF;
(* Rung L739 *)
%WW654 := %UW0.10.8;
(* ----------------------------------------RIGHT DAMPER CONTROL LOGIC----------------------------- *)
(* Rung L743 *)
damperon := STATE3 OR STATE4;
(* Rung L745 *)
IF %MX1 AND SUMMER AND damperon THEN
    TEMPLOWLIM := TEMPSV - %WW132;
    TEMPMAX := TEMPSV + %WW130;
    TEMPE1 := TEMPPV - TEMPLOWLIM;
    %WW420 := %WW132 + %WW130;
    %WW422 := 4000 / %WW420;
    E1 := TEMPE1 * %WW422;
    _t28 := TEMPPV >= TEMPMAX;
END_IF;
%MX16 := _t28;
IF _t28 THEN %UW0.9.7 := 16#FA0; END_IF;
IF %MX1 AND SUMMER AND damperon THEN _t29 := TEMPPV <= TEMPLOWLIM; END_IF;
%MX17 := _t29;
IF _t29 THEN %UW0.9.7 := 16#0; END_IF;
IF %MX1 AND SUMMER AND damperon AND NOT %MX16 AND NOT %MX17 THEN %UW0.9.7 := E1 - 0; END_IF;

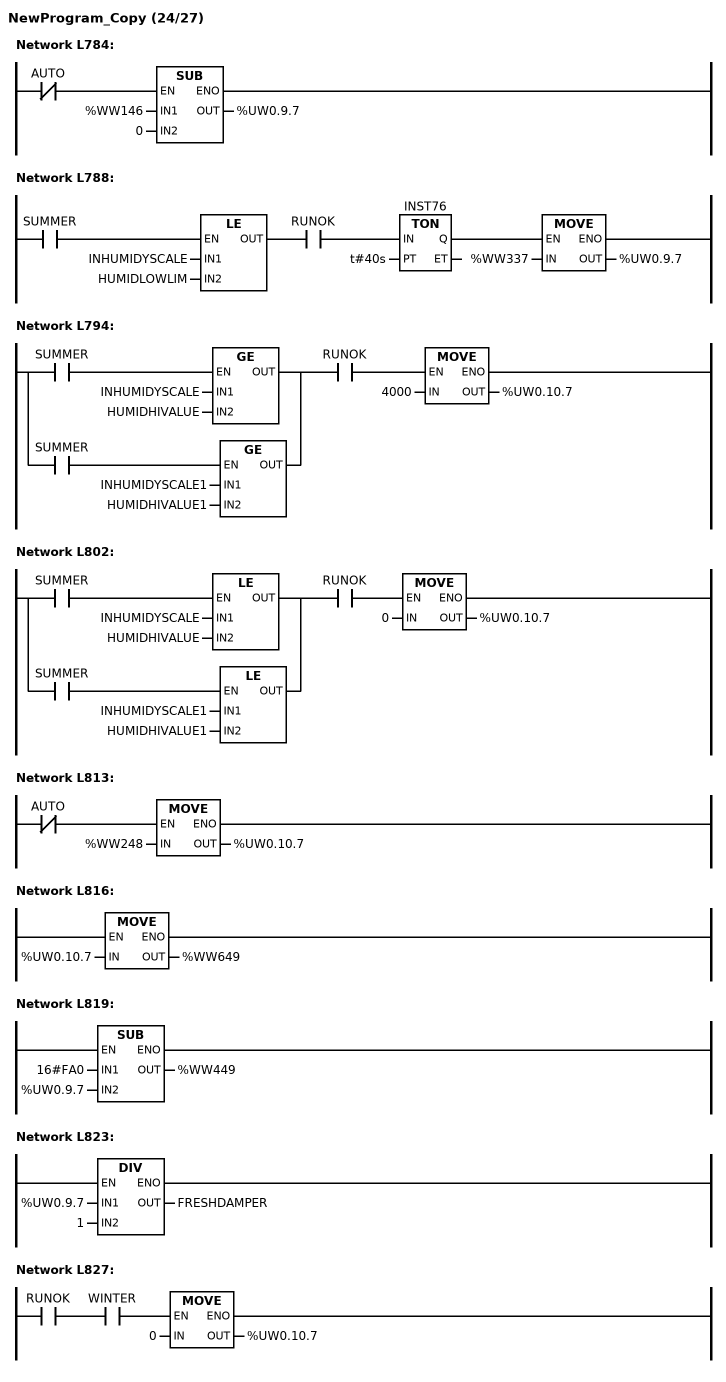
(* Rung L784 *)
IF NOT AUTO THEN %UW0.9.7 := %WW146 - 0; END_IF;
(* Rung L788 *)
IF SUMMER THEN _t30 := INHUMIDYSCALE <= HUMIDLOWLIM; END_IF;
INST76(IN := _t30 AND RUNOK, PT := t#40s);
IF INST76.Q THEN %UW0.9.7 := %WW337; END_IF;
(* Rung L794 *)
IF SUMMER THEN
    _t31 := INHUMIDYSCALE >= HUMIDHIVALUE;
    _t32 := INHUMIDYSCALE1 >= HUMIDHIVALUE1;
END_IF;
IF (_t31 OR _t32) AND RUNOK THEN %UW0.10.7 := 4000; END_IF;
(* Rung L802 *)
IF SUMMER THEN
    _t33 := INHUMIDYSCALE <= HUMIDHIVALUE;
    _t34 := INHUMIDYSCALE1 <= HUMIDHIVALUE1;
END_IF;
IF (_t33 OR _t34) AND RUNOK THEN %UW0.10.7 := 0; END_IF;
(* Rung L813 *)
IF NOT AUTO THEN %UW0.10.7 := %WW248; END_IF;
(* Rung L816 *)
%WW649 := %UW0.10.7;
(* Rung L819 *)
%WW449 := 16#FA0 - %UW0.9.7;
(* Rung L823 *)
FRESHDAMPER := %UW0.9.7 / 1;
(* Rung L827 *)
IF RUNOK AND WINTER THEN %UW0.10.7 := 0; END_IF;

